Fanuc KAREL source: kt00446.KL

PROGRAM KT00446
%STACKSIZE=65535
%PRIORITY=65535
%NOLOCKGROUP
VAR
S1 : STRING[80]
S2 : STRING[80]
OUT : BOOLEAN
BEGIN
S1='A'
S2='B'
S1='A'
S2='B'
-- UNRESOLVED_PC line 12 opcodes [73 73 88 23] marker_code=56
END KT00446
